TYPE ST_Recipe_Cleaning :
STRUCT
	sName					:STRING[80];
	stInfo					:ST_RecipeInfo;
	stPhase					:ARRAY[0..20] OF ST_Cleaning_Phases;
	iType					:INT; 
	iActivePhase			:INT;
END_STRUCT
END_TYPE

(* stored: Version 1.1.0.1
   DUT ST_Recipe_Cleaning: Id {5a33ab64-2a17-4636-9650-9656d83c4f6a} *)
